Staubli VAL3: stop.pgx

program stop()
begin
  cls()
  popUpMsg("Program completed")
  resetMotion()
end
